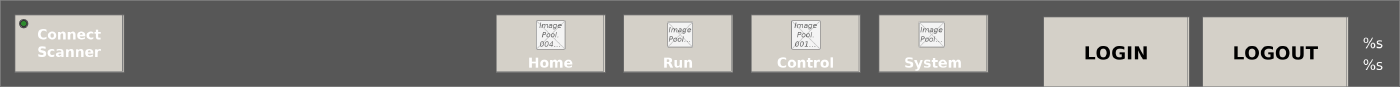
VISUALIZATION FOOTER  // 1920x120
    Textfield (1700,70 200x40), "%s", text variable: MAIN.fb_TimeStamp.SystemDate
    Textfield (1700,40 200x40), "%s", text variable: MAIN.fb_TimeStamp.SystemTime
    Group (855,20 150x80)
        OnMouseClick: change screen: PAGE_RUN
        Button (0,0 150x80), "Run"
        Image (60,10 35x35), image: ImagePool.003-play-button-arrowhead
    Group (1030,20 150x80)
        OnMouseClick: change screen: PAGE_CONTROL
        Button (0,0 150x80), "Control"
        Image (55,8 40x40), image: ImagePool.001-gear
    Group (680,20 150x80)
        OnMouseClick: change screen: PAGE_HOME
        Button (0,0 150x80), "Home"
        Image (55,8 40x40), image: ImagePool.004-home
    Group (1205,20 150x80)
        OnMouseClick: change screen: PAGE_SYSTEM
        Button (0,0 150x80), "System"
        Image (55,10 35x35), image: ImagePool.002-folder
    Button (20,20 150x80), "Connect Scanner"
    Lamp1 (25,25 15x15), style: Lamp-Lamp1-Green
    Group (1431,23 293x60)
        Button (218,0 200x100), "LOGOUT"
            OnMouseClick: VisuUserMgmt Type=Logout
        Button (0,0 200x100), "LOGIN"
            OnMouseClick: VisuUserMgmt Type=Login
END_VISUALIZATION

(* stored: Version 1.1.0.1, ProductVersion 3.1.4024.12
   Visu FOOTER: Id {6c813e44-5918-4dcf-a72e-704131e66eb3} *)
